Yaskawa INFORM job: SKRZYNIA_5540_-90_STOPNI_20BR.JBI

/JOB
//NAME SKRZYNIA_5540_-90_STOPNI_20BR
///FOLDERNAME 02-SKRZYNIE_JOBS
//POS
///NPOS 569,569,0,38,0,0
///TOOL 0
///POSTYPE PULSE
///PULSE
C00000=0,-52280,40443,0,6876,0
C00001=-82314,-24956,17040,-59626,-27382,-6248
C00002=-93910,-8625,17040,-59626,-43355,-6248
C00003=-98846,-1061,-42166,-80308,-57081,16120
C00004=-100452,6057,-48127,-85711,-56704,21322
C00005=-95817,31791,-34187,-84788,-63710,26674
C00006=-95573,33077,-33257,-84645,-64023,26851
C00007=-94315,33778,-32137,-85160,-63467,26714
C00008=-95573,33077,-33257,-84645,-64023,26851
C00009=-94948,31301,-36075,-85235,-63717,27152
C00010=-95573,33077,-33257,-84645,-64023,26851
C00011=-95263,33142,-33256,-84677,-63995,26850
C00012=-95263,33142,-33256,-84677,-63995,26850
C00013=-94230,33719,-32331,-85099,-63538,26735
C00014=-95263,33142,-33256,-84677,-63995,26850
C00015=-94794,31816,-35365,-85120,-63763,27076
C00016=-95263,33142,-33256,-84677,-63995,26850
C00017=-95260,33144,-33256,-84678,-63995,26850
C00018=-95260,33144,-33256,-84678,-63995,26850
C00019=-94260,33701,-32361,-85086,-63552,26738
C00020=-95260,33144,-33256,-84678,-63995,26850
C00021=-94835,31943,-35167,-85080,-63786,27056
C00022=-95260,33144,-33256,-84678,-63995,26850
C00023=-95258,25631,32269,-66559,-75499,2416
C00024=-95258,25631,32269,-66559,-75499,2416
C00025=-94256,26435,33444,-66420,-74940,2208
C00026=-95258,25631,32269,-66559,-75499,2416
C00027=-94857,24030,29962,-66606,-75105,2539
C00028=-95258,25631,32269,-66559,-75499,2416
C00029=-98811,21047,-15512,-99242,-81394,20987
C00030=-98811,21047,-15512,-99242,-81394,20987
C00031=-97856,21592,-14760,-99539,-80803,20995
C00032=-98811,21047,-15512,-99242,-81394,20987
C00033=-98487,19855,-17143,-99373,-81250,21110
C00034=-98811,21047,-15512,-99242,-81394,20987
C00035=-99077,36985,67047,-90824,-74996,11
C00036=-99077,36985,67047,-90824,-74996,11
C00037=-98126,38026,68808,-90519,-74354,-175
C00038=-99077,36985,67047,-90824,-74996,11
C00039=-98675,34279,62554,-90994,-74807,523
C00040=-99077,36985,67047,-90824,-74996,11
C00041=-98046,30065,45001,-99674,-75008,5996
C00042=-96663,27244,32711,-106417,-76052,10001
C00043=-96035,27733,33435,-106407,-75606,10011
C00044=-96663,27244,32711,-106417,-76052,10001
C00045=-96274,25568,30264,-106516,-75947,10234
C00046=-96663,27244,32711,-106417,-76052,10001
C00047=-93416,-2088,4699,-99676,-50441,9343
C00048=-88080,-20128,-3199,-80943,-31244,2335
C00049=-48287,-55439,-44481,-48508,-5390,-10469
C00050=-48287,-44591,-17414,-16172,-14532,-25809
C00051=-73855,-32171,-5678,-43952,-33220,-11069
C00052=-84843,-2315,38096,-46044,-43440,-11681
C00053=-99590,25338,21334,-81459,-78469,-3358
C00054=-99590,25338,21334,-81459,-78469,-3358
C00055=-98681,25943,22203,-81468,-77867,-3455
C00056=-99590,25338,21334,-81459,-78469,-3358
C00057=-99296,24016,19444,-81525,-78239,-3225
C00058=-99590,25338,21334,-81459,-78469,-3358
C00059=-99820,26032,21623,-82067,-78848,-4447
C00060=-99820,26032,21623,-82067,-78848,-4447
C00061=-98898,26645,22513,-82083,-78237,-4546
C00062=-99820,26032,21623,-82067,-78848,-4447
C00063=-99438,24292,19129,-82156,-78552,-4268
C00064=-99820,26032,21623,-82067,-78848,-4447
C00065=-95331,1432,-9864,-84798,-60031,-3557
C00066=-91210,-11403,-27677,-113165,-52408,5733
C00067=-98271,-15326,-41207,-114268,-59488,7673
C00068=-83743,-25164,-57719,-138536,-50905,17366
C00069=-83743,-25361,-52011,-136459,-47698,15842
C00070=-93071,-30029,-62286,-132724,-54351,14554
C00071=-61872,-66272,-83954,-148251,-32298,21081
C00072=-61872,-49557,-32264,-110357,-15428,1928
C00073=-65143,-26385,24751,-20080,-56896,-30933
C00074=-90244,4395,51028,-38516,-59607,-23032
C00075=-79356,-9150,9683,-42499,-40407,-18801
C00076=-98951,25836,42573,-74290,-75705,-4216
C00077=-99097,30513,38864,-76423,-80199,-875
C00078=-97872,31473,40332,-76298,-79437,-1085
C00079=-99097,30513,38864,-76423,-80199,-875
C00080=-98774,28880,36400,-76469,-79893,-679
C00081=-99097,30513,38864,-76423,-80199,-875
C00082=-99862,24525,29609,-86160,-76987,1407
C00083=-99452,22245,7122,-97683,-80070,9369
C00084=-99292,23987,9562,-97373,-81102,9104
C00085=-98184,24694,10564,-97522,-80343,9095
C00086=-99292,23987,9562,-97373,-81102,9104
C00087=-99030,22873,7999,-97442,-80972,9229
C00088=-99292,23987,9562,-97373,-81102,9104
C00089=-95017,-9844,-333,-79976,-47193,-2364
C00090=-62804,-32782,1918,-36164,-30925,-23493
C00091=-48283,-21883,28214,-25170,-26491,48363
C00092=-45951,-10962,51022,-17493,-32991,44756
C00093=-50347,-18571,12268,-49104,-16423,60029
C00094=-52008,-16476,13921,-52720,-16985,61589
C00095=-50839,-15356,14836,-51561,-16264,61168
C00096=-51137,-15647,14596,-51864,-16447,61279
C00097=-52695,-14846,15261,-54465,-17168,62360
C00098=-51384,-16746,13703,-51673,-16698,61154
C00099=-50347,-18571,12268,-49104,-16423,60029
C00100=-52476,-17044,12146,-55476,-16783,62883
C00101=-51467,-16091,12918,-54586,-16145,62570
C00102=-51762,-16375,12685,-54854,-16332,62665
C00103=-53129,-15664,13268,-57063,-16995,63582
C00104=-52557,-17119,12084,-55547,-16837,62908
C00105=-50509,-19000,10610,-51503,-15997,61182
C00106=-52966,-16930,12240,-56194,-17032,63176
C00107=-51879,-15912,13067,-55265,-16346,62852
C00108=-52154,-16175,12851,-55507,-16521,62938
C00109=-53227,-15612,13314,-57215,-17042,63646
C00110=-52966,-16930,12240,-56194,-17032,63176
C00111=-50703,-18403,11066,-52155,-16024,61477
C00112=-52780,-17619,11680,-55562,-17015,62889
C00113=-51306,-16241,12790,-54268,-16084,62435
C00114=-51660,-16583,12512,-54593,-16308,62551
C00115=-53327,-15718,13220,-57282,-17114,63667
C00116=-52780,-17619,11680,-55562,-17015,62889
C00117=-50704,-18401,11069,-52157,-16021,61478
C00118=-53191,-17342,11901,-56260,-17204,63181
C00119=-51773,-16022,12969,-55050,-16305,62760
C00120=-52146,-16378,12679,-55379,-16540,62876
C00121=-53214,-15820,13135,-57085,-17059,63584
C00122=-53002,-17172,12037,-56105,-17083,63128
C00123=-51005,-17995,11387,-52847,-16122,61778
C00124=-52654,-17319,11922,-55560,-16911,62904
C00125=-51372,-16113,12897,-54432,-16099,62508
C00126=-51648,-16379,12679,-54684,-16273,62598
C00127=-52952,-15703,13233,-56807,-16903,63480
C00128=-53323,-17134,12070,-56539,-17248,63304
C00129=-52826,-20105,4812,-63938,-15678,66983
C00130=-52298,-19620,5183,-63681,-15322,66914
C00131=-51076,-18450,6096,-63049,-14499,66733
C00132=-51419,-18785,5831,-63233,-14731,66786
C00133=-52680,-18133,6347,-65138,-15424,67581
C00134=-52924,-19431,7025,-60935,-16175,65505
C00135=-51752,-18759,10786,-53484,-16613,62002
C00136=-52244,-17884,11471,-54682,-16766,62529
C00137=-50303,-16031,12961,-52880,-15542,61887
C00138=-50741,-16464,12607,-53310,-15818,62044
C00139=-52416,-15612,13306,-56135,-16617,63223
C00140=-51898,-18011,11369,-54129,-16600,62301
C00141=-50945,-18019,11363,-52741,-16103,61737
C00142=-51347,-17395,11856,-53690,-16237,62152
C00143=-49990,-16073,12923,-52376,-15383,61677
C00144=-50384,-16465,12603,-52769,-15629,61822
C00145=-52066,-15616,13298,-55654,-16423,63028
C00146=-51792,-17610,11685,-54205,-16494,62350
C00147=-50945,-18019,11363,-52741,-16103,61737
C00148=-50845,-17493,11778,-52895,-15987,61824
C00149=-49521,-16191,12826,-51571,-15155,61341
C00150=-49894,-16567,12520,-51958,-15389,61484
C00151=-51728,-15654,13268,-55171,-16246,62832
C00152=-51082,-17431,11827,-53280,-16102,61986
C00153=-50028,-23690,-6096,-22921,-31075,54538
C00154=-50346,-22995,-5584,-23393,-31002,54768
C00155=-48843,-21430,-4410,-21901,-30270,54078
C00156=-49178,-21788,-4683,-22239,-30433,54235
C00157=-50538,-21100,-4158,-23908,-30654,55032
C00158=-50252,-22811,-5450,-23315,-30936,54734
C00159=-49763,-24818,-32918,-23163,-28604,59699
C00160=-49144,-24298,-32242,-22455,-28505,59304
C00161=-47766,-22458,-30816,-21237,-27774,58615
C00162=-48099,-22913,-31171,-21534,-27949,58786
C00163=-49602,-21997,-30448,-23301,-28174,59772
C00164=-49259,-23869,-32392,-22880,-28141,59533
C00165=-50713,-12366,-58367,-41124,-17813,74400
C00166=-50097,-11438,-57505,-40749,-17495,74109
C00167=-49105,-9842,-55994,-40096,-16991,73614
C00168=-49355,-10250,-56383,-40269,-17116,73742
C00169=-50506,-9357,-55529,-41571,-17503,74586
C00170=-49771,-10920,-57018,-40545,-17327,73951
C00171=-50713,-12366,-58367,-41124,-17813,74400
C00172=-50097,-11438,-57505,-40749,-17495,74109
C00173=-49105,-9842,-55994,-40096,-16991,73614
C00174=-49355,-10250,-56383,-40269,-17116,73742
C00175=-50506,-9357,-55529,-41571,-17503,74586
C00176=-49771,-10920,-57018,-40545,-17327,73951
C00177=-46548,-30139,-39639,-20061,-27197,57955
C00178=-48797,-26670,-6576,-20404,-32539,53259
C00179=-45389,-28224,4312,-35967,-15579,54278
C00180=-40154,-51179,-915,-24203,-8234,36524
C00181=0,-52280,40443,0,6876,0
C00182=-2117,-50103,-33543,-4117,45077,85249
C00183=26439,-48928,-33543,-4117,-52362,85249
C00184=26439,-27355,-33543,-41485,-52362,85249
C00185=39218,-24492,-41653,-51934,-39374,86964
C00186=38244,-2284,-24157,-56964,-37300,90090
C00187=26640,586,-20198,-77712,-51919,89712
C00188=26323,460,-20341,-77681,-52125,89737
C00189=25607,3186,-17293,-77585,-52601,89760
C00190=26323,460,-20341,-77681,-52125,89737
C00191=27719,1044,-19697,-77798,-51218,89644
C00192=26640,586,-20198,-77712,-51919,89712
C00193=46457,7101,-11330,-26648,-40775,82885
C00194=47439,8350,-9833,-26106,-40556,82449
C00195=46334,10684,-6981,-26557,-41070,82837
C00196=47439,8350,-9833,-26106,-40556,82449
C00197=48354,9159,-8854,-25603,-40343,82046
C00198=47439,8350,-9833,-26106,-40556,82449
C00199=24760,-3019,-10726,-94610,-54398,89614
C00200=25145,-1220,-8811,-94681,-54143,89655
C00201=24492,1290,-6066,-94601,-54582,89624
C00202=25145,-1220,-8811,-94681,-54143,89655
C00203=26584,-669,-8211,-94866,-53174,89734
C00204=25145,-1220,-8811,-94681,-54143,89655
C00205=14532,-15164,-22494,-92943,-61192,88617
C00206=-33377,-12679,-20251,-90012,-93751,87621
C00207=-32674,-7309,22058,-70557,-98373,80594
C00208=20046,-29908,-41690,-58842,-55822,75080
C00209=46158,10269,-6164,-23128,-46470,70172
C00210=51306,10256,-19432,-23475,-33025,71236
C00211=50386,12004,-17260,-23922,-33430,71616
C00212=51306,10256,-19432,-23475,-33025,71236
C00213=51995,10928,-18601,-23012,-32906,70879
C00214=51306,10256,-19432,-23475,-33025,71236
C00215=50667,8104,-22050,-23976,-33027,71608
C00216=27434,3323,14960,-56922,-57501,78346
C00217=29014,6574,18756,-56344,-56678,77965
C00218=28326,9009,21700,-56459,-57175,78009
C00219=29014,6574,18756,-56344,-56678,77965
C00220=30292,7183,19486,-55908,-55969,77693
C00221=29014,6574,18756,-56344,-56678,77965
C00222=24457,-1296,-8898,-94600,-54606,89622
C00223=24457,-1296,-8898,-94600,-54606,89622
C00224=23939,748,-6672,-94541,-54956,89598
C00225=24457,-1296,-8898,-94600,-54606,89622
C00226=25626,-864,-8432,-94748,-53818,89684
C00227=24457,-1296,-8898,-94600,-54606,89622
C00228=22058,-20035,-26567,-93333,-56013,88551
C00229=-28907,-25632,-31027,-90338,-90583,86609
C00230=-23923,-11573,-19230,-90501,-87328,87840
C00231=-8646,-8251,-7782,-76032,-82054,83740
C00232=42001,26537,64712,-25019,-74648,68382
C00233=42692,25604,59505,-25067,-71864,68798
C00234=42100,27723,62792,-25233,-72628,68820
C00235=42692,25604,59505,-25067,-71864,68798
C00236=43179,26157,60355,-24838,-71882,68629
C00237=42692,25604,59505,-25067,-71864,68798
C00238=42064,17796,48100,-25604,-70267,69397
C00239=28113,-7386,-15136,-95790,-47335,90009
C00240=28228,-6488,-14240,-95859,-47266,90053
C00241=27767,-5044,-12775,-95858,-47588,90072
C00242=28228,-6488,-14240,-95859,-47266,90053
C00243=29468,-5989,-13737,-96077,-46438,90154
C00244=28228,-6488,-14240,-95859,-47266,90053
C00245=51937,664,-7429,-160484,-50080,89770
C00246=52345,1107,-6938,-160727,-50007,89930
C00247=51359,2767,-5080,-160136,-50147,89540
C00248=52345,1107,-6938,-160727,-50007,89930
C00249=53054,1752,-6222,-161147,-49882,90209
C00250=52345,1107,-6938,-160727,-50007,89930
C00251=51937,664,-7429,-160484,-50080,89770
C00252=29691,-10745,-18393,-95770,-46230,89933
C00253=26663,-19279,-25970,-94307,-48104,89008
C00254=29542,-7588,-14846,-100915,-46930,90773
C00255=29616,-6902,-10165,-96183,-45225,84004
C00256=29097,-5391,-8640,-96201,-45588,84023
C00257=29616,-6902,-10165,-96183,-45225,84004
C00258=31098,-6282,-9543,-96410,-44233,84135
C00259=29616,-6902,-10165,-96183,-45225,84004
C00260=7576,-30273,-44451,-97512,-61182,86443
C00261=-18624,-40022,-50597,-93591,-78329,83668
C00262=-32134,-30783,-37092,-96173,-88064,83581
C00263=23774,-1324,-8929,-94512,-55065,89585
C00264=23774,-1324,-8929,-94512,-55065,89585
C00265=23319,517,-6924,-94461,-55372,89567
C00266=23774,-1324,-8929,-94512,-55065,89585
C00267=25077,-853,-8421,-94674,-54188,89653
C00268=23774,-1324,-8929,-94512,-55065,89585
C00269=22107,-1052,28039,-94807,-51389,77849
C00270=19995,-16885,24938,-75612,-39910,62837
///LIMIT ON
C00271=8393,-42921,36369,-24238,-5473,19544
///LIMIT OFF
C00272=0,-52280,40443,0,6876,0
C00273=-82314,-24956,17040,-59626,-27382,-6248
C00274=-93910,-8625,17040,-59626,-43355,-6248
C00275=-98846,-1061,-42166,-80308,-57081,16120
C00276=-100452,6057,-48127,-85711,-56704,21322
C00277=-95564,34698,-34234,-85516,-63941,27819
C00278=-94021,36658,-30981,-84167,-64832,27454
C00279=-93851,36773,-30815,-84181,-64812,27439
C00280=-95564,34698,-34234,-85516,-63941,27819
C00281=-96930,32282,-32252,-82595,-65816,26305
C00282=-93901,32995,-31122,-83953,-64436,26132
C00283=-93891,32978,-31150,-83961,-64431,26134
C00284=-96930,32282,-32252,-82595,-65816,26305
C00285=-97719,-4194,-31542,-76086,-54596,10626
C00286=-88377,-34186,-45291,-67238,-52212,2442
C00287=-73560,-62084,7826,-28695,-34737,-3666
C00288=0,-52280,40443,0,6876,0
C00289=0,-52280,40443,0,6876,0
C00290=-2117,-50103,-33543,-4117,45077,85249
C00291=26439,-48928,-33543,-4117,-52362,85249
C00292=26439,-27355,-33543,-41485,-52362,85249
C00293=39218,-24492,-41653,-51934,-39374,86964
C00294=37381,-5106,-22608,-53943,-39515,88347
C00295=38119,-10689,-19379,-70548,-34101,88029
C00296=37906,-14512,-22901,-69984,-34376,87713
C00297=41414,6981,-5927,-33889,-45598,86373
C00298=42289,10624,-1511,-33365,-45508,85956
C00299=42351,10656,-1473,-33340,-45486,85935
C00300=41414,6981,-5927,-33889,-45598,86373
C00301=53221,-12364,-8957,-19277,-47766,73858
C00302=11365,-15171,10010,-30164,-77975,82960
C00303=16156,-38280,11293,-23671,-42998,42040
C00304=11365,-47379,10010,-30164,3063,681
C00305=0,-52280,40443,0,6876,0
C00306=0,-36700,24612,42871,-31823,33862
C00307=-44403,-30110,7154,-24155,-23805,45557
C00308=-51570,-19542,10947,-41619,-21811,53396
C00309=-51570,-17239,16856,-38066,-23574,51584
C00310=-55052,-13712,19754,-43494,-24529,53873
C00311=-55190,-12778,21730,-42693,-25060,53437
C00312=-40431,-28773,9158,-17648,-23273,42875
C00313=0,-36700,24612,42871,-31823,33862
C00314=0,-52280,40443,0,6876,0
C00315=0,-52280,40443,0,6876,0
C00316=-73560,-62084,7826,-28695,-34737,-3666
C00317=-88377,-34186,-45291,-67238,-52212,2442
C00318=-99860,-8392,-35780,-75647,-56000,10650
C00319=-100432,21324,12575,-83706,-77956,7498
C00320=-100432,21324,12575,-83706,-77956,7498
C00321=-97477,24790,17443,-83584,-77881,7143
C00322=-97548,25214,18044,-83537,-78171,7107
C00323=-100432,21324,12575,-83706,-77956,7498
C00324=-100473,21504,12824,-83696,-77986,7482
C00325=-97708,25565,18549,-83502,-78342,7077
C00326=-97720,26100,19317,-83456,-78605,7025
C00327=-100432,21324,12575,-83706,-77956,7498
C00328=-98403,3681,-8965,-86029,-63956,7946
C00329=-98851,2841,7216,-80537,-62817,1838
C00330=-99868,-33,22146,-72719,-59601,-5126
C00331=-99028,-10516,17309,-71061,-60695,-4227
C00332=-58820,-39124,10926,-53325,-41870,-3759
C00333=0,-52280,40443,0,6876,0
C00334=-37281,-50778,-9546,-79570,-75313,71156
C00335=-21038,-23698,-30323,-82948,-81132,85647
C00336=-21230,-24252,-33397,-84866,-81311,86227
C00337=26224,-11477,-22521,-89106,-49066,87170
C00338=30473,789,4724,-68168,-47848,79016
C00339=30460,-1091,-3608,-71823,-46530,81583
C00340=26224,-11477,-22521,-89106,-49066,87170
C00341=1250,-26379,-34995,-85812,-66036,85728
C00342=-29373,-17697,-13794,-84248,-87305,82376
C00343=-12562,-22815,-22029,-52123,-75138,85349
C00344=41964,2536,-13642,-34848,-42769,74522
C00345=37974,4101,-26304,-58477,-36842,84551
C00346=37992,4823,-31618,-63468,-34913,87461
C00347=41439,5489,-14791,-37032,-40569,75962
C00348=38833,-3286,10682,-41231,-51577,69207
C00349=-9276,-22918,-17698,-90837,-69000,78700
C00350=-8172,-56778,-49528,-75726,-40055,75711
C00351=-3982,-61001,-53003,-69042,-33087,73336
C00352=37287,-55159,35520,-2191,5667,2084
C00353=0,-52280,40443,0,6876,0
C00354=0,-36700,24612,42871,-31823,33862
C00355=-44403,-30110,7154,-24155,-23805,45557
C00356=-44403,-30110,7154,-24155,-23805,45557
C00357=-42101,-12213,25656,-103795,-5192,78630
C00358=-46259,-8171,27719,-110365,-8144,81138
C00359=-67532,2461,52564,-58221,-38014,54436
C00360=-67092,2390,52438,-57975,-37749,54380
C00361=-61158,-4651,8765,-137237,-40004,88174
C00362=-56934,-15752,2926,-132390,-27589,90381
C00363=-47073,-34549,9488,-27883,-30316,51458
C00364=0,-52280,40443,0,6876,0
C00365=0,-52280,40443,0,6876,0
C00366=-73560,-62084,7826,-28695,-34737,-3666
C00367=-96366,-17217,16860,-56620,-71703,-18245
C00368=-98152,-14905,2044,-65675,-67485,-3494
C00369=-100467,-7393,-15195,-81625,-60158,6002
C00370=-99336,18440,8642,-84276,-74234,7647
C00371=-99336,18440,8642,-84276,-74234,7647
C00372=-97907,25479,18429,-83510,-78268,7080
C00373=-97774,25771,18838,-83486,-78362,7054
C00374=-99336,18440,8642,-84276,-74234,7647
C00375=-99336,20364,19482,-82786,-74642,4774
C00376=-98337,25059,18813,-87846,-78771,10707
C00377=-98337,23926,10585,-88652,-78855,12971
C00378=-99528,19847,13673,-83665,-74506,6500
C00379=-89817,-17341,-38408,-97132,-45323,12250
C00380=-100347,-21961,-42251,-93939,-52125,11121
C00381=-60204,-59872,-73451,-117647,-17639,18840
C00382=-37721,-67612,11381,-1325,-438,-7850
C00383=0,-52280,40443,0,6876,0
C00384=37287,-55159,35520,-2191,5667,2084
C00385=40042,-68802,-18337,-47708,-19461,45384
C00386=16481,-63411,-38742,-86271,-37962,67106
C00387=28646,-23138,-32952,-89786,-42552,85395
C00388=38882,-16596,-17625,-44304,-41043,72768
C00389=40930,-6862,-13364,-47045,-37020,74415
C00390=41744,-3361,-9781,-46774,-36492,74231
C00391=41678,-4243,-16493,-50979,-33997,76666
C00392=40930,-6862,-13364,-47045,-37020,74415
C00393=38882,-16596,-17625,-44304,-41043,72768
C00394=28646,-23138,-32952,-89786,-42552,85395
C00395=29905,-15291,-26411,-91102,-43435,86304
C00396=31540,-7654,-19248,-92177,-42391,86919
C00397=31445,-8095,-22888,-97196,-43117,89457
C00398=29637,-16450,-35189,-96198,-44206,89682
C00399=-7164,-46429,-55577,-86274,-68578,84143
C00400=40042,-68802,-18337,-47708,-19461,45384
C00401=37287,-55159,35520,-2191,5667,2084
C00402=0,-52280,40443,0,6876,0
C00403=-37164,-60659,6466,-13301,-5027,19773
C00404=-45362,-39990,2831,-27538,-17767,40935
C00405=-57189,-26834,-7130,-38780,-31731,51561
C00406=-55974,-20661,-3180,-39617,-29741,52134
C00407=-55991,-28453,-45977,-64163,-20900,63765
C00408=-57189,-26834,-7130,-38780,-31731,51561
C00409=-41180,-61187,4729,-17280,-8498,23442
C00410=0,-52280,40443,0,6876,0
C00411=0,-52280,40443,0,6876,0
C00412=-43180,-50572,-20637,-6552,-29302,-38834
C00413=-79425,-37128,-15462,-51820,-35721,-18807
C00414=-93702,-21743,-5664,-65079,-41536,-12324
C00415=-94876,-11469,-23586,-124528,-59237,5423
C00416=-92861,23404,17376,-116518,-76732,-1573
C00417=-96665,29896,42633,-98437,-75635,-11031
C00418=-96665,37701,65506,-96077,-73868,-15674
C00419=-98256,26642,30161,-104402,-77650,-7294
C00420=-94876,-11469,-23586,-124528,-59237,5423
C00421=-94108,-26192,-19530,-80749,-38523,-6311
C00422=-79425,-37128,-15462,-51820,-35721,-18807
C00423=-44920,-50063,-20090,-8739,-29356,-37564
C00424=-37721,-67612,11381,-1325,-438,-7850
C00425=0,-52280,40443,0,6876,0
C00426=40043,-68802,-18337,-47706,-19461,45383
C00427=27078,-46675,7729,-35821,-60236,53359
C00428=37661,6027,34279,-36092,-58837,68690
C00429=38848,9668,32452,-36978,-55195,69693
C00430=45203,15557,41040,-24527,-60177,66840
C00431=37661,2340,23735,-37788,-55306,70200
C00432=22173,-30639,7984,-58136,-45615,60133
C00433=37287,-55159,35520,-2191,5667,2084
C00434=0,-52280,40443,0,6876,0
C00435=-23708,-46776,23536,-16027,-4787,19738
C00436=-50917,-40459,4132,-34421,-18173,42391
C00437=-54964,-26842,8528,-44141,-23181,52038
C00438=-51719,-20944,8196,-48593,-18539,54728
C00439=-53338,-16066,12564,-52314,-18938,56375
C00440=-53668,-14237,17353,-48629,-20286,54493
C00441=-18010,-41727,-5437,24633,-20435,23511
C00442=-18010,-41727,-5437,24633,-20435,23511
C00443=-43180,-50572,-20637,-6552,-29302,-38834
C00444=-37721,-67612,11381,-1325,-438,-7850
C00445=0,-52280,40443,0,6876,0
C00446=-7830,-25136,17099,-55306,-64068,52084
C00447=34592,-23156,18291,-29932,-45204,43222
C00448=27626,-5609,7480,-74303,-46810,69713
C00449=30162,-7263,-3756,-79871,-43922,73611
C00450=30945,-3557,12,-79972,-43367,73694
C00451=30934,-3652,-86,-79966,-43372,73693
C00452=29106,-7674,-4162,-79972,-44640,73655
C00453=-2837,-32019,-23857,-80741,-66785,72567
C00454=9534,-43450,13514,-26959,-29486,38723
C00455=22834,-59963,22946,-6692,-2150,9612
C00456=0,-52280,40443,0,6876,0
C00457=-23708,-46776,23536,-16027,-4787,19738
C00458=-50917,-40459,4132,-34421,-18173,42391
C00459=-51059,-36587,4608,-36647,-19418,45358
C00460=-50113,-22729,10834,-36393,-23396,50963
C00461=-57831,-20321,-874,-74195,-20905,72937
C00462=-57885,-15500,12470,-61600,-22854,66553
C00463=-50113,-22729,10834,-36393,-23396,50963
C00464=-45969,-44671,-42317,80322,10570,10889
C00465=-31285,-69981,-10849,-7246,-6842,20992
C00466=0,-52280,40443,0,6876,0
C00467=-37721,-67612,11381,-1325,-438,-7850
C00468=-43180,-50572,-20637,-6552,-29302,-38834
C00469=-92181,-6909,34626,-50562,-49190,-21840
C00470=-101117,-5694,-18308,-85789,-60825,2377
C00471=-97622,-3602,-16155,-86160,-58465,2400
C00472=-99754,24347,18348,-83049,-78046,1543
C00473=-98401,23935,17754,-83131,-77323,1564
C00474=-98274,24050,17917,-83129,-77329,1551
C00475=-99954,24418,19993,-82828,-78557,1051
C00476=-99712,24798,18984,-83012,-78332,1506
C00477=-99852,25442,19906,-82977,-78439,1439
C00478=-98294,26390,21274,-82926,-78604,1336
C00479=-98320,27540,23370,-82787,-79202,1083
C00480=-99852,25442,19906,-82977,-78439,1439
C00481=-99768,8894,-2445,-89351,-68751,3793
C00482=-96099,-3787,-16815,-92200,-58195,4535
C00483=-97559,-25159,-36085,-93407,-46496,3918
C00484=-68601,-52593,-52127,-95725,-25602,3235
C00485=-80632,-38079,-20908,-64053,-45216,-12949
C00486=-43180,-50572,-20637,-6552,-29302,-38834
///LIMIT ON
C00487=-37721,-67612,11381,-1325,-438,-7850
///LIMIT OFF
C00488=54026,-30203,28811,7745,-28969,5087
C00489=55906,-29650,27841,6704,-28568,42061
C00490=3910,-49110,-20873,-64325,-51391,71742
C00491=9596,-41005,-15480,-61992,-50741,70573
C00492=34629,-5327,8260,-51720,-47880,65426
C00493=35679,2837,17551,-51053,-47466,65038
C00494=35689,-56,7549,-54586,-44718,67469
C00495=34629,-5327,8260,-51720,-47880,65426
C00496=9596,-41005,-15480,-61992,-50741,70573
C00497=29660,-4584,-26917,-122917,-59269,85605
C00498=30458,-1431,-23593,-123278,-58903,85810
C00499=32051,-581,-21149,-126899,-58917,85995
C00500=28378,-5181,-30467,-124970,-61925,86269
C00501=9596,-41005,-15480,-61992,-50741,70573
C00502=4124,-42500,-16101,-63937,-54198,71061
C00503=22834,-59963,22946,-6692,-2150,9612
C00504=0,-52280,40443,0,6876,0
C00505=-44101,-76445,-48847,-15697,-17168,40457
C00506=-48984,-30078,-36716,-21434,-29637,58750
C00507=-50484,-13386,-55713,-36158,-19724,71897
C00508=-50319,-9696,-53018,-37576,-18929,72579
C00509=-57729,15185,-57220,-77412,-21272,89270
C00510=-57753,15208,-57190,-77395,-21282,89267
C00511=-50484,-13386,-55713,-36158,-19724,71897
C00512=-49763,-25421,-36239,-24565,-26935,60445
C00513=-50529,-22709,-3778,-22940,-31995,54502
C00514=-45389,-28224,4312,-35967,-15579,54278
C00515=-40154,-51179,-915,-24203,-8234,36524
C00516=0,-52280,40443,0,6876,0
C00517=0,-52280,40443,0,6876,0
///LIMIT ON
C00518=-37721,-67612,11381,-1325,-438,-7850
///LIMIT OFF
C00519=-43180,-50572,-20637,-6552,-29302,-38834
C00520=-43180,-50572,-20637,-6552,-29302,-38834
C00521=-91233,-13472,9135,-57436,-42793,-15671
C00522=-94453,18451,26397,-64403,-69695,-4898
C00523=-94848,25710,19994,-67599,-74328,1083
C00524=-94734,25454,19627,-67614,-74234,1097
C00525=-94605,24228,10738,-68938,-72404,3439
C00526=-96555,21614,11724,-68276,-72695,2131
C00527=-99000,22482,23037,-75261,-76004,639
C00528=-97210,28604,31066,-74659,-78513,378
C00529=-97154,26647,21384,-75593,-77346,2770
C00530=-100531,16612,13557,-75306,-72509,1088
C00531=-98914,15791,22093,-91892,-69242,2220
C00532=-98524,31242,37673,-92432,-80087,2200
C00533=-98508,35203,51300,-91477,-79539,-794
C00534=-99299,29399,42249,-91532,-77608,155
C00535=-99299,39874,71997,-89061,-76925,-5800
C00536=-98153,38420,66100,-91432,-76531,-4068
C00537=-98147,36464,60868,-91873,-76694,-3060
C00538=-99718,12303,6039,-96207,-71156,6635
C00539=-93032,-8711,-3060,-81304,-48072,-4095
C00540=-98228,-14972,-11291,-81392,-49231,-4002
C00541=-91129,-17870,8831,-66292,-48444,-14183
C00542=-68865,-35989,-5252,-49829,-38105,-21179
C00543=-15566,-52364,-9989,12732,-35649,-46896
C00544=0,-52278,40443,-31822,-65283,46097
C00545=7820,3000,44222,-77356,-66876,70486
C00546=23103,22769,71034,-65639,-61603,67373
C00547=25078,30713,84198,-63240,-61811,65668
C00548=25008,30264,83410,-63369,-61766,65773
C00549=23103,22769,71034,-65639,-61603,67373
C00550=23103,22769,71034,-65639,-61603,67373
C00551=25078,30713,84198,-63240,-61811,65668
C00552=25008,30264,83410,-63369,-61766,65773
C00553=23103,22769,71034,-65639,-61603,67373
C00554=-3014,-20441,-7349,-104591,-68614,79454
C00555=-3014,-20441,-7349,-104591,-68614,79454
C00556=-13238,-21720,-1359,-93359,-59492,72612
C00557=10261,-46634,14475,-36899,-22136,31570
///LIMIT ON
C00558=22834,-59963,22946,-6692,-2150,9612
///LIMIT OFF
C00559=0,-52280,40443,0,6876,0
///LIMIT ON
C00560=-23708,-46776,23536,-16027,-4787,19738
///LIMIT OFF
C00561=-50917,-40459,4132,-34421,-18173,42391
C00562=-49876,-21948,7530,-68838,-10324,59148
C00563=-46721,-18942,9765,-68167,-8197,59205
C00564=-47628,-14741,12915,-75746,-8483,62696
C00565=-48046,-13368,16308,-68442,-9096,59180
C00566=-42573,-24036,4541,-56448,-5917,54155
C00567=-31287,-69981,-10850,-7253,-6843,20996
C00568=0,-52280,40443,0,6876,0
BC00000=471249
BC00001=460491
BC00002=460491
BC00003=460491
BC00004=460491
BC00005=482540
BC00006=483588
BC00007=483588
BC00008=483588
BC00009=483588
BC00010=483588
BC00011=529782
BC00012=529782
BC00013=529782
BC00014=529782
BC00015=529782
BC00016=529782
BC00017=575949
BC00018=575949
BC00019=575949
BC00020=575949
BC00021=575949
BC00022=575949
BC00023=551765
BC00024=551765
BC00025=551765
BC00026=551765
BC00027=551765
BC00028=551765
BC00029=597819
BC00030=597819
BC00031=597819
BC00032=597819
BC00033=597819
BC00034=597819
BC00035=596567
BC00036=596567
BC00037=596567
BC00038=596567
BC00039=596567
BC00040=596567
BC00041=623804
BC00042=642102
BC00043=642102
BC00044=642102
BC00045=642102
BC00046=642102
BC00047=619616
BC00048=619616
BC00049=642599
BC00050=714482
BC00051=745522
BC00052=745522
BC00053=836176
BC00054=836176
BC00055=836176
BC00056=836176
BC00057=836176
BC00058=836176
BC00059=881624
BC00060=881624
BC00061=881624
BC00062=881624
BC00063=881624
BC00064=881624
BC00065=881624
BC00066=887605
BC00067=887605
BC00068=887605
BC00069=887605
BC00070=887605
BC00071=887605
BC00072=887605
BC00073=983293
BC00074=981254
BC00075=985702
BC00076=990046
BC00077=996594
BC00078=996594
BC00079=996594
BC00080=996594
BC00081=996594
BC00082=994630
BC00083=1060317
BC00084=1060317
BC00085=1060317
BC00086=1060317
BC00087=1060317
BC00088=1060317
BC00089=993852
BC00090=983691
BC00091=935062
BC00092=958518
BC00093=1027445
BC00094=1027445
BC00095=1027445
BC00096=1027445
BC00097=1027445
BC00098=1027445
BC00099=964364
BC00100=968743
BC00101=968743
BC00102=968743
BC00103=968743
BC00104=968743
BC00105=903417
BC00106=903417
BC00107=903417
BC00108=903417
BC00109=903417
BC00110=903417
BC00111=846075
BC00112=846075
BC00113=846075
BC00114=846075
BC00115=846075
BC00116=846075
BC00117=780190
BC00118=780190
BC00119=780190
BC00120=780190
BC00121=780190
BC00122=780190
BC00123=722535
BC00124=722535
BC00125=722535
BC00126=722535
BC00127=722535
BC00128=722535
BC00129=657432
BC00130=657432
BC00131=657432
BC00132=657432
BC00133=657432
BC00134=657432
BC00135=600107
BC00136=600107
BC00137=600107
BC00138=600107
BC00139=600107
BC00140=600107
BC00141=534593
BC00142=534593
BC00143=534593
BC00144=534593
BC00145=534593
BC00146=534593
BC00147=477174
BC00148=477174
BC00149=477174
BC00150=477174
BC00151=477174
BC00152=477174
BC00153=474905
BC00154=474905
BC00155=474905
BC00156=474905
BC00157=474905
BC00158=474905
BC00159=474905
BC00160=474905
BC00161=474905
BC00162=474905
BC00163=474905
BC00164=474905
BC00165=474905
BC00166=474905
BC00167=474905
BC00168=474905
BC00169=474905
BC00170=474905
BC00171=428822
BC00172=428822
BC00173=428822
BC00174=428822
BC00175=428822
BC00176=428822
BC00177=474905
BC00178=474905
BC00179=474901
BC00180=548577
BC00181=548577
BC00182=423885
BC00183=423885
BC00184=423885
BC00185=423885
BC00186=423885
BC00187=423882
BC00188=423882
BC00189=423882
BC00190=423882
BC00191=423882
BC00192=423882
BC00193=517447
BC00194=516208
BC00195=516208
BC00196=516208
BC00197=516208
BC00198=516208
BC00199=462401
BC00200=462401
BC00201=462401
BC00202=462401
BC00203=462401
BC00204=462401
BC00205=462401
BC00206=462401
BC00207=581968
BC00208=647467
BC00209=647467
BC00210=647467
BC00211=647467
BC00212=647467
BC00213=647467
BC00214=647467
BC00215=647467
BC00216=600589
BC00217=600589
BC00218=600589
BC00219=600589
BC00220=600589
BC00221=600589
BC00222=646713
BC00223=646713
BC00224=646713
BC00225=646713
BC00226=646713
BC00227=646713
BC00228=646713
BC00229=646713
BC00230=703926
BC00231=764819
BC00232=734650
BC00233=734650
BC00234=734650
BC00235=734650
BC00236=734650
BC00237=734650
BC00238=734650
BC00239=762000
BC00240=762000
BC00241=762000
BC00242=762000
BC00243=762000
BC00244=762000
BC00245=768744
BC00246=768744
BC00247=768744
BC00248=768744
BC00249=768744
BC00250=768744
BC00251=768744
BC00252=762000
BC00253=762000
BC00254=869424
BC00255=869424
BC00256=869424
BC00257=869424
BC00258=869424
BC00259=869424
BC00260=869424
BC00261=869424
BC00262=983898
BC00263=992364
BC00264=992364
BC00265=992364
BC00266=992364
BC00267=992364
BC00268=992364
BC00269=927243
BC00270=910363
BC00271=869677
BC00272=473857
BC00273=460491
BC00274=460491
BC00275=460491
BC00276=460491
BC00277=491299
BC00278=491278
BC00279=483675
BC00280=491299
BC00281=530690
BC00282=530690
BC00283=523662
BC00284=530690
BC00285=557568
BC00286=557568
BC00287=557568
BC00288=542207
BC00289=492150
BC00290=423885
BC00291=423885
BC00292=423885
BC00293=423885
BC00294=418215
BC00295=406365
BC00296=406365
BC00297=507950
BC00298=507950
BC00299=500226
BC00300=507950
BC00301=493160
BC00302=493160
BC00303=493160
BC00304=493160
BC00305=493160
BC00306=598171
BC00307=670543
BC00308=729889
BC00309=728141
BC00310=728141
BC00311=789114
BC00312=789114
BC00313=598171
BC00314=556285
BC00315=557568
BC00316=557568
BC00317=557568
BC00318=606305
BC00319=559125
BC00320=474638
BC00321=474638
BC00322=467026
BC00323=474638
BC00324=536109
BC00325=536109
BC00326=543656
BC00327=536109
BC00328=539958
BC00329=628234
BC00330=599778
BC00331=599778
BC00332=599778
BC00333=599778
BC00334=542360
BC00335=599440
BC00336=482963
BC00337=482963
BC00338=482963
BC00339=482963
BC00340=482963
BC00341=482963
BC00342=482963
BC00343=633179
BC00344=633182
BC00345=633182
BC00346=633182
BC00347=633182
BC00348=590162
BC00349=577838
BC00350=565789
BC00351=612529
BC00352=620193
BC00353=620193
BC00354=828164
BC00355=903144
BC00356=942427
BC00357=909055
BC00358=930245
BC00359=950170
BC00360=1007113
BC00361=1029951
BC00362=961342
BC00363=868420
BC00364=557568
BC00365=557568
BC00366=528880
BC00367=572227
BC00368=592163
BC00369=606305
BC00370=587350
BC00371=582221
BC00372=582227
BC00373=588358
BC00374=582221
BC00375=641167
BC00376=648252
BC00377=646780
BC00378=643131
BC00379=650479
BC00380=650479
BC00381=648520
BC00382=733103
BC00383=733103
BC00384=620193
BC00385=620193
BC00386=625652
BC00387=635598
BC00388=635598
BC00389=635598
BC00390=635598
BC00391=635598
BC00392=635598
BC00393=635598
BC00394=635598
BC00395=658627
BC00396=658630
BC00397=665879
BC00398=658627
BC00399=658627
BC00400=620193
BC00401=620193
BC00402=620193
BC00403=561542
BC00404=498768
BC00405=467432
BC00406=467432
BC00407=467432
BC00408=467432
BC00409=539526
BC00410=539526
BC00411=748464
BC00412=748464
BC00413=630778
BC00414=630772
BC00415=630772
BC00416=630772
BC00417=638952
BC00418=638952
BC00419=636403
BC00420=630772
BC00421=630772
BC00422=652282
BC00423=713933
BC00424=733103
BC00425=733103
BC00426=667407
BC00427=721208
BC00428=721208
BC00429=721208
BC00430=727232
BC00431=730010
BC00432=686453
BC00433=620193
BC00434=620193
BC00435=576077
BC00436=557154
BC00437=596115
BC00438=604917
BC00439=604794
BC00440=662711
BC00441=664655
BC00442=784947
BC00443=795297
BC00444=733103
BC00445=733103
BC00446=727492
BC00447=727492
BC00448=759331
BC00449=759331
BC00450=759331
BC00451=766564
BC00452=759331
BC00453=759331
BC00454=672725
BC00455=672725
BC00456=672725
BC00457=766882
BC00458=806462
BC00459=818228
BC00460=851878
BC00461=860102
BC00462=909902
BC00463=851878
BC00464=813387
BC00465=767805
BC00466=733103
BC00467=733103
BC00468=748464
BC00469=748464
BC00470=831036
BC00471=832865
BC00472=832865
BC00473=832865
BC00474=839696
BC00475=839696
BC00476=877964
BC00477=878266
BC00478=878754
BC00479=885787
BC00480=878266
BC00481=840209
BC00482=834137
BC00483=827396
BC00484=765830
BC00485=798734
BC00486=810658
BC00487=748464
BC00488=762701
BC00489=765633
BC00490=830967
BC00491=835024
BC00492=852883
BC00493=852883
BC00494=852883
BC00495=852883
BC00496=835024
BC00497=861491
BC00498=861491
BC00499=861491
BC00500=861491
BC00501=835024
BC00502=835024
BC00503=672725
BC00504=672725
BC00505=543617
BC00506=474905
BC00507=474905
BC00508=474905
BC00509=459544
BC00510=450616
BC00511=474905
BC00512=474905
BC00513=474905
BC00514=474901
BC00515=548577
BC00516=548577
BC00517=748464
BC00518=748464
BC00519=869948
BC00520=986791
BC00521=981739
BC00522=1008171
BC00523=1008171
BC00524=1008171
BC00525=1008171
BC00526=1008171
BC00527=1008171
BC00528=1008171
BC00529=1008171
BC00530=1006011
BC00531=1030226
BC00532=1030226
BC00533=1030226
BC00534=1030226
BC00535=1030226
BC00536=1030226
BC00537=1042625
BC00538=1042625
BC00539=995149
BC00540=992199
BC00541=972060
BC00542=967683
BC00543=967683
BC00544=921533
BC00545=921533
BC00546=946591
BC00547=946591
BC00548=953713
BC00549=946591
BC00550=997282
BC00551=997282
BC00552=1004404
BC00553=997282
BC00554=1013986
BC00555=963295
BC00556=908449
BC00557=770245
BC00558=688086
BC00559=688086
BC00560=577701
BC00561=467723
BC00562=467723
BC00563=467723
BC00564=467723
BC00565=526528
BC00566=527247
BC00567=757643
BC00568=757643
///POSTYPE BASE
///RECTAN
///RCONF 0,0,0,0,0,0,0,0,0,0,0,0,0,0,0,0,0,0,0,0,0,0,0,0
P00006=-2.449,0.031,8.825,0.0000,0.0000,0.0000
///RCONF 1,0,0,0,0,0,0,0,0,0,0,0,0,0,0,0,0,0,0,0,0,0,0,0
P00300=-0.036,-1.505,2.318,0.0000,0.0000,0.0000
///RCONF 0,0,0,0,0,0,0,0,0,0,0,0,0,0,0,0,0,0,0,0,0,0,0,0
P00301=0.005,-4.708,-4.628,0.0000,0.0000,0.0000
P00302=0.052,-2.937,-4.426,0.0000,0.0000,0.0000
P00303=-0.004,-1.437,-4.584,0.0000,0.0000,0.0000
P00304=0.028,-1.666,-4.234,0.0000,0.0000,0.0000
P00305=-0.003,-1.920,-3.501,0.0000,0.0000,0.0000
P00306=0.015,-2.252,-3.054,0.0000,0.0000,0.0000
P00308=-0.003,-2.092,-4.888,0.0000,0.0000,0.0000
P00309=-0.040,-2.205,-4.992,0.0000,0.0000,0.0000
P00311=-0.007,-2.079,-5.307,0.0000,0.0000,0.0000
P00312=-0.032,2.202,-7.632,0.0000,0.0000,0.0000
///RCONF 1,0,0,0,0,0,0,0,0,0,0,0,0,0,0,0,0,0,0,0,0,0,0,0
P00349=0.060,0.167,-1.133,0.0000,0.0000,0.0000
///RCONF 0,0,0,0,0,0,0,0,0,0,0,0,0,0,0,0,0,0,0,0,0,0,0,0
P00350=11.519,-0.008,1.149,0.0000,0.0000,0.0000
P00351=13.563,-0.027,-0.653,0.0000,0.0000,0.0000
P00352=13.252,-0.027,-0.827,0.0000,0.0000,0.0000
P00353=10.971,-0.082,0.776,0.0000,0.0000,0.0000
P00354=-0.024,2.508,-1.824,0.0000,0.0000,0.0000
P00355=-0.001,2.528,-1.131,0.0000,0.0000,0.0000
P00356=-0.034,2.921,-0.262,0.0000,0.0000,0.0000
P00357=0.003,3.386,-0.091,0.0000,0.0000,0.0000
P00358=0.014,3.037,-0.020,0.0000,0.0000,0.0000
P00359=-0.005,2.731,0.912,0.0000,0.0000,0.0000
P00360=-0.011,3.412,0.438,0.0000,0.0000,0.0000
P00361=0.018,3.050,1.253,0.0000,0.0000,0.0000
P00362=0.014,2.784,0.148,0.0000,0.0000,0.0000
P00400=5.920,-3.503,-0.024,0.0000,0.0000,0.0000
P00401=3.430,-0.021,1.131,0.0000,0.0000,0.0000
P00402=-0.253,1.107,3.062,0.0000,0.0000,0.0000
P00403=-3.666,-0.015,5.328,0.0000,0.0000,0.0000
///RCONF 1,0,0,0,0,0,0,0,0,0,0,0,0,0,0,0,0,0,0,0,0,0,0,0
P00404=0.029,4.189,-1.030,0.0000,0.0000,0.0000
///RCONF 0,0,0,0,0,0,0,0,0,0,0,0,0,0,0,0,0,0,0,0,0,0,0,0
P00405=2.420,0.007,1.427,0.0000,0.0000,0.0000
P00406=3.513,-0.022,0.429,0.0000,0.0000,0.0000
///RCONF 1,0,0,0,1,0,0,0,0,0,0,0,0,0,0,0,0,0,0,0,0,0,0,0
P00407=-0.029,2.348,-1.469,0.0000,0.0000,0.0000
P00408=0.010,1.346,-1.479,0.0000,0.0000,0.0000
///RCONF 1,0,0,0,0,0,0,0,0,0,0,0,0,0,0,0,0,0,0,0,0,0,0,0
P00409=-0.026,2.090,-1.483,0.0000,0.0000,0.0000
P00410=0.001,4.491,-0.583,0.0000,0.0000,0.0000
///RCONF 1,0,0,0,1,0,0,0,0,0,0,0,0,0,0,0,0,0,0,0,0,0,0,0
P00411=-0.015,3.627,0.872,0.0000,0.0000,0.0000
//INST
///DATE 2025/02/25 14:00
///ATTR SC,RW
///GROUP1 RB1,BS1
NOP
CALL JOB:MOVE_INTO_TUNNEL
MOVJ C00000 BC00000 VJ=30.00
MOVJ C00001 BC00001 VJ=30.00
MOVJ C00002 BC00002 VJ=30.00
MOVL C00003 BC00003 V=500.0
MOVJ C00004 BC00004 VJ=20.00
'------------------------
'W65.3
'------------------------
MOVL C00005 BC00005 V=333.3
MOVL C00006 BC00006 V=166.7 PL=0
REFP 3 C00007 BC00007
CALL JOB:SEARCH-R1
SET P0300 P0006
SFTON P0300
MOVL C00008 BC00008 V=66.7 PL=0
REFP 3 C00009 BC00009
CALL JOB:SEARCH-R1
SET P0300 P0006
SFTON P0300
MOVL C00010 BC00010 V=66.7 PL=0
SFTOF
'------------------------
'W65.5
'------------------------
MOVL C00011 BC00011 V=500.0
MOVL C00012 BC00012 V=166.7 PL=0
REFP 3 C00013 BC00013
CALL JOB:SEARCH-R1
SET P0301 P0006
SFTON P0301
MOVL C00014 BC00014 V=166.7 PL=0
REFP 3 C00015 BC00015
CALL JOB:SEARCH-R1
SET P0301 P0006
SFTON P0301
MOVL C00016 BC00016 V=166.7 PL=0
SFTOF
'------------------------
'W65.7
'------------------------
MOVL C00017 BC00017 V=500.0
MOVL C00018 BC00018 V=166.7 PL=0
REFP 3 C00019 BC00019
CALL JOB:SEARCH-R1
SET P0302 P0006
SFTON P0302
MOVL C00020 BC00020 V=166.7 PL=0
REFP 3 C00021 BC00021
CALL JOB:SEARCH-R1
SET P0302 P0006
SFTON P0302
MOVL C00022 BC00022 V=166.7 PL=0
SFTOF
'------------------------
'W65.10
'------------------------
MOVL C00023 BC00023 V=500.0
MOVL C00024 BC00024 V=166.7 PL=0
REFP 3 C00025 BC00025
CALL JOB:SEARCH-R1
SET P0303 P0006
SFTON P0303
MOVL C00026 BC00026 V=166.7 PL=0
REFP 3 C00027 BC00027
CALL JOB:SEARCH-R1
SET P0303 P0006
SFTON P0303
MOVL C00028 BC00028 V=166.7 PL=0
SFTOF
'------------------------
'W65.12
'------------------------
MOVL C00029 BC00029 V=500.0
MOVL C00030 BC00030 V=166.7 PL=0
REFP 3 C00031 BC00031
CALL JOB:SEARCH-R1
SET P0304 P0006
SFTON P0304
MOVL C00032 BC00032 V=166.7 PL=0
REFP 3 C00033 BC00033
CALL JOB:SEARCH-R1
SET P0304 P0006
SFTON P0304
MOVL C00034 BC00034 V=166.7 PL=0
SFTOF
'------------------------
'W65.15
'------------------------
MOVL C00035 BC00035 V=333.3
MOVL C00036 BC00036 V=166.7 PL=0
REFP 3 C00037 BC00037
CALL JOB:SEARCH-R1
SET P0305 P0006
SFTON P0305
MOVL C00038 BC00038 V=166.7 PL=0
REFP 3 C00039 BC00039
CALL JOB:SEARCH-R1
SET P0305 P0006
SFTON P0305
MOVL C00040 BC00040 V=166.7 PL=0
SFTOF
'------------------------
'W65.17
'------------------------
MOVL C00041 BC00041 V=333.3
MOVL C00042 BC00042 V=166.7 PL=0
REFP 3 C00043 BC00043
CALL JOB:SEARCH-R1
SET P0306 P0006
SFTON P0306
MOVL C00044 BC00044 V=166.7 PL=0
REFP 3 C00045 BC00045
CALL JOB:SEARCH-R1
SET P0306 P0006
SFTON P0306
MOVL C00046 BC00046 V=166.7 PL=0
SFTOF
MOVL C00047 BC00047 V=333.3
MOVL C00048 BC00048 V=500.0
MOVL C00049 BC00049 V=500.0
MOVJ C00050 BC00050 VJ=50.00
MOVL C00051 BC00051 V=500.0
MOVL C00052 BC00052 V=500.0
'------------------------
'W65.20
'------------------------
'------------------------
MOVL C00053 BC00053 V=333.3
MOVL C00054 BC00054 V=166.7 PL=0
REFP 3 C00055 BC00055
CALL JOB:SEARCH-R1
SET P0308 P0006
SFTON P0308
MOVL C00056 BC00056 V=166.7 PL=0
REFP 3 C00057 BC00057
CALL JOB:SEARCH-R1
SET P0308 P0006
SFTON P0308
MOVL C00058 BC00058 V=166.7 PL=0
SFTOF
'------------------------
'W65.25
'------------------------
MOVL C00059 BC00059 V=500.0
MOVL C00060 BC00060 V=166.7 PL=0
REFP 3 C00061 BC00061
CALL JOB:SEARCH-R1
SET P0309 P0006
SFTON P0309
MOVL C00062 BC00062 V=166.7 PL=0
REFP 3 C00063 BC00063
CALL JOB:SEARCH-R1
SET P0309 P0006
SFTON P0309
MOVL C00064 BC00064 V=166.7 PL=0
SFTOF
MOVL C00065 BC00065 V=166.7
MOVL C00066 BC00066 V=666.7
MOVL C00067 BC00067 V=666.7
MOVL C00068 BC00068 V=666.7
MOVL C00069 BC00069 V=666.7
MOVL C00070 BC00070 V=666.7
MOVL C00071 BC00071 V=666.7
MOVL C00072 BC00072 V=666.7
MOVL C00073 BC00073 V=666.7
MOVL C00074 BC00074 V=666.7
MOVL C00075 BC00075 V=666.7
'------------------------
'W65.28
'------------------------
'W65.30
'------------------------
MOVL C00076 BC00076 V=500.0
MOVL C00077 BC00077 V=166.7 PL=0
REFP 3 C00078 BC00078
CALL JOB:SEARCH-R1
SET P0311 P0006
SFTON P0311
MOVL C00079 BC00079 V=166.7 PL=0
REFP 3 C00080 BC00080
CALL JOB:SEARCH-R1
SET P0311 P0006
SFTON P0311
MOVL C00081 BC00081 V=166.7 PL=0
SFTOF
MOVL C00082 BC00082 V=333.3
MOVL C00083 BC00083 V=333.3
MOVL C00084 BC00084 V=166.7
REFP 3 C00085 BC00085
CALL JOB:SEARCH-R1
SET P0312 P0006
SFTON P0312
MOVL C00086 BC00086 V=166.7 PL=0
REFP 3 C00087 BC00087
CALL JOB:SEARCH-R1
SET P0312 P0006
SFTON P0312
MOVL C00088 BC00088 V=166.7 PL=0
SFTOF
MOVL C00089 BC00089 V=333.3
MOVL C00090 BC00090 V=333.3
MOVJ C00091 BC00091 VJ=30.00
MOVJ C00092 BC00092 VJ=30.00
MOVL C00093 BC00093 V=500.0
SFTOF
MOVL C00094 BC00094 V=166.7 PL=0
REFP 3 C00095 BC00095
CALL JOB:SEARCH-R1
SET P0349 P0006
SFTON P0349
MOVL C00096 BC00096 V=166.7 PL=0
REFP 3 C00097 BC00097
CALL JOB:SEARCH-R1
SET P0349 P0006
SFTON P0349
MOVL C00098 BC00098 V=166.7 PL=0
SFTOF
MOVL C00099 BC00099 V=333.3
SFTOF
'------------------------
'W251A
'------------------------
MOVL C00100 BC00100 V=166.7 PL=0
REFP 3 C00101 BC00101
CALL JOB:SEARCH-R1
SET P0350 P0006
SFTON P0350
MOVL C00102 BC00102 V=166.7 PL=0
REFP 3 C00103 BC00103
CALL JOB:SEARCH-R1
SET P0350 P0006
SFTON P0350
MOVL C00104 BC00104 V=166.7 PL=0
SFTOF
'------------------------
'W254A P
'------------------------
MOVJ C00105 BC00105 VJ=40.00
MOVL C00106 BC00106 V=166.7 PL=0
REFP 3 C00107 BC00107
CALL JOB:SEARCH-R1
SET P0351 P0006
SFTON P0351
MOVL C00108 BC00108 V=166.7 PL=0
REFP 3 C00109 BC00109
CALL JOB:SEARCH-R1
SET P0351 P0006
SFTON P0351
MOVL C00110 BC00110 V=166.7 PL=0
SFTOF
'------------------------
'W254A L
'------------------------
MOVJ C00111 BC00111 VJ=40.00
MOVL C00112 BC00112 V=166.7 PL=0
REFP 3 C00113 BC00113
CALL JOB:SEARCH-R1
SET P0352 P0006
SFTON P0352
MOVL C00114 BC00114 V=166.7 PL=0
REFP 3 C00115 BC00115
CALL JOB:SEARCH-R1
SET P0352 P0006
SFTON P0352
MOVL C00116 BC00116 V=166.7 PL=0
SFTOF
'------------------------
'W250A P
'------------------------
MOVJ C00117 BC00117 VJ=40.00
MOVL C00118 BC00118 V=166.7 PL=0
REFP 3 C00119 BC00119
CALL JOB:SEARCH-R1
SET P0353 P0006
SFTON P0353
MOVL C00120 BC00120 V=66.7 PL=0
REFP 3 C00121 BC00121
CALL JOB:SEARCH-R1
SET P0353 P0006
SFTON P0353
MOVL C00122 BC00122 V=66.7 PL=0
SFTOF
'------------------------
'W250A L
'------------------------
MOVJ C00123 BC00123 VJ=40.00
MOVL C00124 BC00124 V=166.7 PL=0
REFP 3 C00125 BC00125
CALL JOB:SEARCH-R1
SET P0354 P0006
SFTON P0354
MOVL C00126 BC00126 V=66.7 PL=0
REFP 3 C00127 BC00127
CALL JOB:SEARCH-R1
SET P0354 P0006
SFTON P0354
MOVL C00128 BC00128 V=166.7 PL=0
SFTOF
'------------------------
'W253A P
'------------------------
MOVJ C00129 BC00129 VJ=40.00
MOVL C00130 BC00130 V=166.7 PL=0
REFP 3 C00131 BC00131
CALL JOB:SEARCH-R1
SET P0355 P0006
SFTON P0355
MOVL C00132 BC00132 V=166.7 PL=0
REFP 3 C00133 BC00133
CALL JOB:SEARCH-R1
SET P0355 P0006
SFTON P0355
MOVL C00134 BC00134 V=166.7 PL=0
SFTOF
'------------------------
'W253A L
'------------------------
MOVJ C00135 BC00135 VJ=40.00
MOVL C00136 BC00136 V=166.7 PL=0
REFP 3 C00137 BC00137
CALL JOB:SEARCH-R1
SET P0356 P0006
SFTON P0356
MOVL C00138 BC00138 V=166.7 PL=0
REFP 3 C00139 BC00139
CALL JOB:SEARCH-R1
SET P0356 P0006
SFTON P0356
MOVL C00140 BC00140 V=166.7 PL=0
SFTOF
'------------------------
'W256A P
'------------------------
MOVJ C00141 BC00141 VJ=40.00
MOVL C00142 BC00142 V=166.7 PL=0
REFP 3 C00143 BC00143
CALL JOB:SEARCH-R1
SET P0357 P0006
SFTON P0357
MOVL C00144 BC00144 V=166.7 PL=0
REFP 3 C00145 BC00145
CALL JOB:SEARCH-R1
SET P0357 P0006
SFTON P0357
MOVL C00146 BC00146 V=166.7 PL=0
SFTOF
'------------------------
'W256A L
'------------------------
MOVJ C00147 BC00147 VJ=40.00
MOVL C00148 BC00148 V=166.7 PL=0
REFP 3 C00149 BC00149
CALL JOB:SEARCH-R1
SET P0358 P0006
SFTON P0358
MOVL C00150 BC00150 V=166.7 PL=0
REFP 3 C00151 BC00151
CALL JOB:SEARCH-R1
SET P0358 P0006
SFTON P0358
MOVL C00152 BC00152 V=166.7 PL=0
SFTOF
'------------------------
'W252A P
'------------------------
MOVL C00153 BC00153 V=666.7
MOVL C00154 BC00154 V=166.7 PL=0
REFP 3 C00155 BC00155
CALL JOB:SEARCH-R1
SET P0359 P0006
SFTON P0359
MOVL C00156 BC00156 V=166.7 PL=0
REFP 3 C00157 BC00157
CALL JOB:SEARCH-R1
SET P0359 P0006
SFTON P0359
MOVL C00158 BC00158 V=166.7 PL=0
SFTOF
'------------------------
'W252A L
'------------------------
MOVL C00159 BC00159 V=500.0
MOVL C00160 BC00160 V=166.7 PL=0
REFP 3 C00161 BC00161
CALL JOB:SEARCH-R1
SET P0360 P0006
SFTON P0360
MOVL C00162 BC00162 V=166.7 PL=0
REFP 3 C00163 BC00163
CALL JOB:SEARCH-R1
SET P0360 P0006
SFTON P0360
MOVL C00164 BC00164 V=166.7 PL=0
SFTOF
'------------------------
'W255A
'------------------------
MOVL C00165 BC00165 V=500.0
MOVL C00166 BC00166 V=166.7 PL=0
REFP 3 C00167 BC00167
CALL JOB:SEARCH-R1
SET P0361 P0006
SFTON P0361
MOVL C00168 BC00168 V=166.7 PL=0
REFP 3 C00169 BC00169
CALL JOB:SEARCH-R1
SET P0361 P0006
SFTON P0361
MOVL C00170 BC00170 V=166.7 PL=0
SFTOF
MOVL C00171 BC00171 V=500.0
MOVL C00172 BC00172 V=166.7 PL=0
REFP 3 C00173 BC00173
CALL JOB:SEARCH-R1
SET P0362 P0006
SFTON P0362
MOVL C00174 BC00174 V=166.7 PL=0
REFP 3 C00175 BC00175
CALL JOB:SEARCH-R1
SET P0362 P0006
SFTON P0362
MOVL C00176 BC00176 V=166.7 PL=0
SFTOF
MOVL C00177 BC00177 V=666.7
MOVL C00178 BC00178 V=666.7
MOVL C00179 BC00179 V=666.7
MOVJ C00180 BC00180 VJ=40.00
MOVJ C00181 BC00181 VJ=40.00
COMM MOVJ C00182 BC00182 VJ=40.00
COMM MOVJ C00183 BC00183 VJ=40.00
COMM MOVJ C00184 BC00184 VJ=40.00
COMM MOVJ C00185 BC00185 VJ=40.00
COMM MOVJ C00186 BC00186 VJ=30.00
COMM '------------------------
COMM 'W61.3
COMM '------------------------
COMM MOVL C00187 BC00187 V=500.0
COMM MOVL C00188 BC00188 V=166.7 PL=0
COMM REFP 3 C00189 BC00189
COMM CALL JOB:SEARCH-R1
COMM SET P0400 P0006
COMM SFTON P0400
COMM MOVL C00190 BC00190 V=166.7 PL=0
COMM REFP 3 C00191 BC00191
COMM CALL JOB:SEARCH-R1
COMM SET P0400 P0006
COMM SFTON P0400
COMM MOVL C00192 BC00192 V=166.7 PL=0
COMM SFTOF
COMM 'BELKA PRZEJAZD
COMM MOVL C00193 BC00193 V=333.3
COMM '------------------------
COMM 'W61.5
COMM '------------------------
COMM MOVL C00194 BC00194 V=166.7 PL=0
COMM REFP 3 C00195 BC00195
COMM CALL JOB:SEARCH-R1
COMM SET P0401 P0006
COMM SFTON P0401
COMM MOVL C00196 BC00196 V=166.7 PL=0
COMM REFP 3 C00197 BC00197
COMM CALL JOB:SEARCH-R1
COMM SET P0401 P0006
COMM SFTON P0401
COMM MOVL C00198 BC00198 V=166.7 PL=0
COMM SFTOF
COMM '------------------------
COMM 'W61.7
COMM '------------------------
COMM MOVL C00199 BC00199 V=500.0
COMM MOVL C00200 BC00200 V=166.7 PL=0
COMM REFP 3 C00201 BC00201
COMM CALL JOB:SEARCH-R1
COMM SET P0402 P0006
COMM SFTON P0402
COMM MOVL C00202 BC00202 V=166.7 PL=0
COMM REFP 3 C00203 BC00203
COMM CALL JOB:SEARCH-R1
COMM SET P0402 P0006
COMM SFTON P0402
COMM MOVL C00204 BC00204 V=166.7 PL=0
COMM SFTOF
COMM MOVL C00205 BC00205 V=500.0
COMM '------------------------
COMM 'W61.10
COMM '------------------------
COMM MOVJ C00206 BC00206 VJ=30.00
COMM MOVJ C00207 BC00207 VJ=50.00
COMM MOVJ C00208 BC00208 VJ=50.00
COMM MOVL C00209 BC00209 V=500.0
COMM MOVL C00210 BC00210 V=166.7 PL=0
COMM REFP 3 C00211 BC00211
COMM CALL JOB:SEARCH-R1
COMM SET P0403 P0006
COMM SFTON P0403
COMM MOVL C00212 BC00212 V=166.7 PL=0
COMM REFP 3 C00213 BC00213
COMM CALL JOB:SEARCH-R1
COMM SET P0403 P0006
COMM SFTON P0403
COMM MOVL C00214 BC00214 V=166.7 PL=0
COMM SFTOF
COMM MOVL C00215 BC00215 V=333.3
COMM '------------------------
COMM 'W61.12
COMM '------------------------
COMM MOVL C00216 BC00216 V=666.7
COMM MOVL C00217 BC00217 V=166.7 PL=0
COMM REFP 3 C00218 BC00218
COMM CALL JOB:SEARCH-R1
COMM SET P0404 P0006
COMM SFTON P0404
COMM MOVL C00219 BC00219 V=166.7 PL=0
COMM REFP 3 C00220 BC00220
COMM CALL JOB:SEARCH-R1
COMM SET P0404 P0006
COMM SFTON P0404
COMM MOVL C00221 BC00221 V=166.7 PL=0
COMM SFTOF
COMM '------------------------
COMM 'W61.15
COMM '------------------------
COMM MOVL C00222 BC00222 V=666.7
COMM MOVL C00223 BC00223 V=166.7 PL=0
COMM REFP 3 C00224 BC00224
COMM CALL JOB:SEARCH-R1
COMM SET P0405 P0006
COMM SFTON P0405
COMM MOVL C00225 BC00225 V=166.7 PL=0
COMM REFP 3 C00226 BC00226
COMM CALL JOB:SEARCH-R1
COMM SET P0405 P0006
COMM SFTON P0405
COMM MOVL C00227 BC00227 V=166.7 PL=0
COMM SFTOF
COMM MOVL C00228 BC00228 V=666.7
COMM MOVJ C00229 BC00229 VJ=50.00
COMM MOVJ C00230 BC00230 VJ=50.00
COMM MOVJ C00231 BC00231 VJ=50.00
COMM '------------------------
COMM 'W61.17
COMM '------------------------
COMM MOVL C00232 BC00232 V=416.7
COMM MOVL C00233 BC00233 V=166.7 PL=0
COMM REFP 3 C00234 BC00234
COMM CALL JOB:SEARCH-R1
COMM SET P0406 P0006
COMM SFTON P0406
COMM MOVL C00235 BC00235 V=166.7 PL=0
COMM REFP 3 C00236 BC00236
COMM CALL JOB:SEARCH-R1
COMM SET P0406 P0006
COMM SFTON P0406
COMM MOVL C00237 BC00237 V=166.7 PL=0
COMM SFTOF
COMM MOVL C00238 BC00238 V=333.3
COMM '------------------------
COMM 'W61.20
COMM '------------------------
COMM MOVL C00239 BC00239 V=666.7
COMM MOVL C00240 BC00240 V=166.7 PL=0
COMM REFP 3 C00241 BC00241
COMM CALL JOB:SEARCH-R1
COMM SET P0407 P0006
COMM SFTON P0407
COMM MOVL C00242 BC00242 V=166.7 PL=0
COMM REFP 3 C00243 BC00243
COMM CALL JOB:SEARCH-R1
COMM SET P0407 P0006
COMM SFTON P0407
COMM MOVL C00244 BC00244 V=166.7 PL=0
COMM SFTOF
COMM '------------------------
COMM 'W61.23
COMM '------------------------
COMM MOVL C00245 BC00245 V=500.0
COMM MOVL C00246 BC00246 V=166.7 PL=0
COMM REFP 3 C00247 BC00247
COMM CALL JOB:SEARCH-R1
COMM SET P0408 P0006
COMM SFTON P0408
COMM MOVL C00248 BC00248 V=166.7 PL=0
COMM REFP 3 C00249 BC00249
COMM CALL JOB:SEARCH-R1
COMM SET P0408 P0006
COMM SFTON P0408
COMM MOVL C00250 BC00250 V=166.7 PL=0
COMM SFTOF
COMM MOVL C00251 BC00251 V=333.3
COMM MOVL C00252 BC00252 V=666.7
COMM MOVL C00253 BC00253 V=666.7
COMM '------------------------
COMM 'W61.25
COMM '------------------------
COMM MOVL C00254 BC00254 V=500.0
COMM MOVL C00255 BC00255 V=166.7 PL=0
COMM REFP 3 C00256 BC00256
COMM CALL JOB:SEARCH-R1
COMM SET P0409 P0006
COMM SFTON P0409
COMM MOVL C00257 BC00257 V=166.7 PL=0
COMM REFP 3 C00258 BC00258
COMM CALL JOB:SEARCH-R1
COMM SET P0409 P0006
COMM SFTON P0409
COMM MOVL C00259 BC00259 V=166.7 PL=0
COMM SFTOF
COMM MOVL C00260 BC00260 V=666.7
COMM MOVJ C00261 BC00261 VJ=50.00
COMM MOVJ C00262 BC00262 VJ=50.00
COMM GETE D040 P0409 (1)
COMM GETE D041 P0409 (2)
COMM GETE D042 P0409 (3)
COMM SETE P0410 (1) D040
COMM SETE P0410 (2) D041
COMM SETE P0410 (3) D042
COMM '------------------------
COMM 'W61.30
COMM '------------------------
COMM MOVL C00263 BC00263 V=500.0
COMM MOVL C00264 BC00264 V=166.7 PL=0
COMM REFP 3 C00265 BC00265
COMM CALL JOB:SEARCH-R1
COMM SET P0411 P0006
COMM SFTON P0411
COMM MOVL C00266 BC00266 V=166.7 PL=0
COMM REFP 3 C00267 BC00267
COMM CALL JOB:SEARCH-R1
COMM SET P0411 P0006
COMM SFTON P0411
COMM MOVL C00268 BC00268 V=166.7 PL=0
COMM SFTOF
COMM MOVL C00269 BC00269 V=666.7
COMM MOVJ C00270 BC00270 VJ=50.00
MOVJ C00271 BC00271 VJ=70.00
CALL JOB:FRONT_SEARCH_-90ST-2_5540
MOVJ C00272 BC00272 VJ=60.00
MOVJ C00273 BC00273 VJ=50.00
MOVJ C00274 BC00274 VJ=50.00
MOVL C00275 BC00275 V=666.7
MOVJ C00276 BC00276 VJ=30.00
'------------------------
'W65.3
'------------------------
SFTON P0300
MOVL C00277 BC00277 V=333.3
MOVL C00278 BC00278 V=166.7 PL=0
MACRO1 MJ#(0) ARGF10
ARCON
MOVL C00279 BC00279 V=10.8
ARCOF
MOVL C00280 BC00280 V=166.7
SFTOF
'------------------------
'W65.5
'------------------------
SFTON P0301
MOVL C00281 BC00281 V=666.7
MOVL C00282 BC00282 V=166.7 PL=0
MACRO1 MJ#(0) ARGF9
ARCON
MOVL C00283 BC00283 V=8.3
ARCOF
MOVL C00284 BC00284 V=166.7
SFTOF
MOVL C00285 BC00285 V=500.0
MOVL C00286 BC00286 V=666.7
MOVJ C00287 BC00287 VJ=40.00
COMM MOVJ C00288 BC00288 VJ=60.00
COMM '::::::::::::::::::::::::::::::::
COMM '::::::::::::::::::::::::::::::::
COMM '::::::::::::::::::::::::::::::::
COMM '::::::::::::::::::::::::::::::::
COMM '::::::::::::::::::::::::::::::::
COMM MOVJ C00289 BC00289 VJ=50.00
COMM MOVJ C00290 BC00290 VJ=50.00
COMM MOVJ C00291 BC00291 VJ=40.00
COMM MOVJ C00292 BC00292 VJ=40.00
COMM MOVJ C00293 BC00293 VJ=40.00
COMM MOVJ C00294 BC00294 VJ=40.00
COMM MOVL C00295 BC00295 V=666.7
COMM '------------------------
COMM 'W61.3
COMM '------------------------
COMM SFTON P0400
COMM ARCOF
COMM MOVL C00296 BC00296 V=500.0
COMM SFTOF
COMM 'BELKA PRZEJAZD
COMM '------------------------
COMM 'W61.5
COMM '------------------------
COMM SFTON P0401
COMM MOVL C00297 BC00297 V=666.7
COMM MOVL C00298 BC00298 V=166.7 PL=0
COMM MACRO1 MJ#(0) ARGF24
COMM ARCON
COMM MOVL C00299 BC00299 V=7.5
COMM ARCOF
COMM MOVL C00300 BC00300 V=250.0
COMM SFTOF
COMM MOVL C00301 BC00301 V=500.0
COMM MOVJ C00302 BC00302 VJ=40.00
COMM MOVJ C00303 BC00303 VJ=40.00
COMM MOVJ C00304 BC00304 VJ=50.00
COMM MOVJ C00305 BC00305 VJ=50.00
MOVJ C00306 BC00306 VJ=50.00
MOVJ C00307 BC00307 VJ=50.00
MOVL C00308 BC00308 V=666.7
'------------------------
'W250A
'------------------------
SFTON P0354
MOVL C00309 BC00309 V=666.7
MOVL C00310 BC00310 V=166.7 PL=0
MACRO1 MJ#(0) ARGF9
ARCON
SFTOF
SFTON P0353
MOVL C00311 BC00311 V=11.7
ARCOF
MOVL C00312 BC00312 V=333.3
SFTOF
MOVJ C00313 BC00313 VJ=50.00
MOVJ C00314 BC00314 VJ=60.00
MOVJ C00315 BC00315 VJ=40.00
MOVJ C00316 BC00316 VJ=50.00
MOVJ C00317 BC00317 VJ=40.00
MOVJ C00318 BC00318 VJ=30.00
MOVJ C00319 BC00319 VJ=15.00
'------------------------
'W65.7
'------------------------
SFTON P0302
MOVL C00320 BC00320 V=833.3
MOVL C00321 BC00321 V=166.7 PL=0
MACRO1 MJ#(0) ARGF10
ARCON
MOVL C00322 BC00322 V=10.8
ARCOF
MOVL C00323 BC00323 V=166.7
SFTOF
'------------------------
'W65.10
'------------------------
SFTON P0303
MOVL C00324 BC00324 V=666.7
MOVL C00325 BC00325 V=166.7 PL=0
ARCON
MOVL C00326 BC00326 V=10.8
ARCOF
MOVL C00327 BC00327 V=166.7
SFTOF
MOVL C00328 BC00328 V=333.3
MOVL C00329 BC00329 V=666.7
MOVJ C00330 BC00330 VJ=30.00
MOVJ C00331 BC00331 VJ=30.00
MOVJ C00332 BC00332 VJ=30.00
MOVJ C00333 BC00333 VJ=50.00
COMM '::::::::::::::::::::::::::::::::
COMM '::::::::::::::::::::::::::::::::
COMM '------------------------
COMM 'W61.7
COMM '------------------------
COMM '::::::::::::::::::::::::::::::::
COMM '::::::::::::::::::::::::::::::::
COMM MOVJ C00334 BC00334 VJ=30.00
COMM MOVJ C00335 BC00335 VJ=30.00
COMM MOVJ C00336 BC00336 VJ=40.00
COMM SFTON P0402
COMM MOVL C00337 BC00337 V=500.0
COMM MOVL C00338 BC00338 V=166.7 PL=0
COMM MACRO1 MJ#(0) ARGF24
COMM ARCON
COMM MOVL C00339 BC00339 V=7.5
COMM ARCOF
COMM MOVL C00340 BC00340 V=250.0
COMM SFTOF
COMM MOVJ C00341 BC00341 VJ=30.00
COMM MOVJ C00342 BC00342 VJ=40.00
COMM MOVJ C00343 BC00343 VJ=50.00
COMM '------------------------
COMM 'W61.10
COMM '------------------------
COMM SFTON P0403
COMM MOVL C00344 BC00344 V=500.0
COMM MOVL C00345 BC00345 V=166.7 PL=0
COMM MACRO1 MJ#(0) ARGF24
COMM ARCON
COMM MOVL C00346 BC00346 V=7.5
COMM ARCOF
COMM MOVL C00347 BC00347 V=250.0
COMM SFTOF
COMM MOVL C00348 BC00348 V=500.0
COMM MOVL C00349 BC00349 V=666.7
COMM MOVL C00350 BC00350 V=666.7
COMM MOVJ C00351 BC00351 VJ=50.00
COMM MOVJ C00352 BC00352 VJ=50.00
COMM MOVJ C00353 BC00353 VJ=50.00
COMM '::::::::::::::::::::::::
COMM '::::::::::::::::::::::::
COMM '::::::::::::::::::::::::
COMM '::::::::::::::::::::::::
COMM '::::::::::::::::::::::::
COMM '::::::::::::::::::::::::
COMM '::::::::::::::::::::::::
MOVJ C00354 BC00354 VJ=50.00
MOVJ C00355 BC00355 VJ=50.00
MOVJ C00356 BC00356 VJ=50.00
'------------------------
'W251B
'------------------------
MOVL C00357 BC00357 V=500.0
MOVL C00358 BC00358 V=500.0
SFTON P0350
MOVL C00359 BC00359 V=166.7 PL=0
MACRO1 MJ#(0) ARGF9
ARCON
SFTOF
SFTON P0349
MOVL C00360 BC00360 V=11.3
MOVL C00361 BC00361 V=11.3
ARCOF
MOVL C00362 BC00362 V=333.3
SFTOF
MOVJ C00363 BC00363 VJ=50.00
MOVJ C00364 BC00364 VJ=50.00
MOVJ C00365 BC00365 VJ=10.00
MOVJ C00366 BC00366 VJ=50.00
MOVJ C00367 BC00367 VJ=50.00
MOVJ C00368 BC00368 VJ=25.00
MOVJ C00369 BC00369 VJ=20.00
MOVJ C00370 BC00370 VJ=20.00
'------------------------
'W65.12
'------------------------
SFTON P0304
MOVL C00371 BC00371 V=333.3
MOVL C00372 BC00372 V=166.7 PL=0
MACRO1 MJ#(0) ARGF10
ARCON
MOVL C00373 BC00373 V=10.8
ARCOF
MOVL C00374 BC00374 V=166.7
SFTOF
'------------------------
'W65.15
'------------------------
SFTON P0305
MOVL C00375 BC00375 V=666.7
MOVL C00376 BC00376 V=166.7 PL=0
MACRO1 MJ#(0) ARGF9
ARCON
MOVL C00377 BC00377 V=10.8
ARCOF
MOVL C00378 BC00378 V=200.0
SFTOF
MOVL C00379 BC00379 V=250.0
MOVL C00380 BC00380 V=416.7
MOVL C00381 BC00381 V=666.7
COMM MOVJ C00382 BC00382 VJ=50.00
COMM MOVJ C00383 BC00383 VJ=50.00
COMM '::::::::::::::::::::::::
COMM '::::::::::::::::::::::::
COMM '::::::::::::::::::::::::
COMM '::::::::::::::::::::::::
COMM '::::::::::::::::::::::::
COMM '::::::::::::::::::::::::
COMM '::::::::::::::::::::::::
COMM MOVJ C00384 BC00384 VJ=50.00
COMM MOVJ C00385 BC00385 VJ=50.00
COMM MOVJ C00386 BC00386 VJ=50.00
COMM '::::::::::::::::::::::::::::::::
COMM '::::::::::::::::::::::::::::::::
COMM '------------------------
COMM 'W61.12
COMM '------------------------
COMM '::::::::::::::::::::::::::::::::
COMM '::::::::::::::::::::::::::::::::
COMM MOVL C00387 BC00387 V=833.3
COMM MOVL C00388 BC00388 V=666.7
COMM MOVL C00389 BC00389 V=500.0
COMM SFTON P0404
COMM MOVL C00390 BC00390 V=166.7 PL=0
COMM MACRO1 MJ#(0) ARGF24
COMM ARCON
COMM MOVL C00391 BC00391 V=6.7
COMM ARCOF
COMM MOVL C00392 BC00392 V=333.3
COMM SFTOF
COMM MOVL C00393 BC00393 V=500.0
COMM MOVL C00394 BC00394 V=666.7
COMM '------------------------
COMM 'W61.15
COMM '------------------------
COMM SFTON P0405
COMM MOVL C00395 BC00395 V=666.7
COMM MOVL C00396 BC00396 V=166.7 PL=0
COMM MACRO1 MJ#(0) ARGF24
COMM ARCON
COMM MOVL C00397 BC00397 V=6.7
COMM ARCOF
COMM MOVL C00398 BC00398 V=250.0
COMM SFTOF
COMM MOVJ C00399 BC00399 VJ=40.00
COMM MOVJ C00400 BC00400 VJ=40.00
COMM MOVJ C00401 BC00401 VJ=40.00
COMM MOVJ C00402 BC00402 VJ=40.00
COMM '::::::::::::::::::::::::
COMM '::::::::::::::::::::::::
COMM '::::::::::::::::::::::::
COMM '::::::::::::::::::::::::
COMM '::::::::::::::::::::::::
COMM '::::::::::::::::::::::::
COMM '::::::::::::::::::::::::
COMM MOVJ C00403 BC00403 VJ=40.00
COMM MOVJ C00404 BC00404 VJ=40.00
COMM '------------------------
COMM 'W252B
COMM '------------------------
SFTON P0359
MOVL C00405 BC00405 V=666.7
MOVL C00406 BC00406 V=166.7 PL=0
MACRO1 MJ#(0) ARGF9
ARCON
SFTOF
SFTON P0358
MOVL C00407 BC00407 V=10.8
ARCOF
MOVL C00408 BC00408 V=250.0
SFTOF
MOVJ C00409 BC00409 VJ=50.00
MOVJ C00410 BC00410 VJ=50.00
MOVJ C00411 BC00411 VJ=60.00
MOVJ C00412 BC00412 VJ=40.00
MOVJ C00413 BC00413 VJ=30.00
MOVL C00414 BC00414 V=500.0
MOVL C00415 BC00415 V=333.3
'------------------------
'W65.17
'------------------------
SFTON P0306
MOVL C00416 BC00416 V=333.3
MOVL C00417 BC00417 V=166.7 PL=0
MACRO1 MJ#(0) ARGF10
ARCON
MOVL C00418 BC00418 V=10.8
ARCOF
MOVL C00419 BC00419 V=166.7
SFTOF
MOVL C00420 BC00420 V=333.3
MOVL C00421 BC00421 V=500.0
MOVL C00422 BC00422 V=500.0
MOVJ C00423 BC00423 VJ=40.00
COMM MOVJ C00424 BC00424 VJ=60.00
COMM MOVJ C00425 BC00425 VJ=60.00
COMM '::::::::::::::::::::::::
COMM '::::::::::::::::::::::::
COMM '::::::::::::::::::::::::
COMM '::::::::::::::::::::::::
COMM '::::::::::::::::::::::::
COMM '::::::::::::::::::::::::
COMM '::::::::::::::::::::::::
COMM MOVJ C00426 BC00426 VJ=60.00
COMM '::::::::::::::::::::::::::::::::
COMM '::::::::::::::::::::::::::::::::
COMM '------------------------
COMM 'W61.17
COMM '------------------------
COMM '::::::::::::::::::::::::::::::::
COMM '::::::::::::::::::::::::::::::::
COMM SFTON P0406
COMM MOVJ C00427 BC00427 VJ=40.00
COMM MOVL C00428 BC00428 V=500.0
COMM MOVL C00429 BC00429 V=166.7 PL=0
COMM MACRO1 MJ#(0) ARGF24
COMM ARCON
COMM MOVL C00430 BC00430 V=6.7
COMM ARCOF
COMM MOVL C00431 BC00431 V=333.3
COMM SFTOF
COMM MOVJ C00432 BC00432 VJ=30.00
COMM MOVJ C00433 BC00433 VJ=40.00
COMM MOVJ C00434 BC00434 VJ=50.00
COMM '------------------------
COMM 'W253A
'------------------------
COMM MOVJ C00435 BC00435 VJ=50.00
MOVJ C00436 BC00436 VJ=50.00
SFTON P0356
MOVL C00437 BC00437 V=500.0
MOVL C00438 BC00438 V=500.0
MOVL C00439 BC00439 V=166.7 PL=0
MACRO1 MJ#(0) ARGF9
ARCON
SFTOF
SFTON P0355
MOVL C00440 BC00440 V=11.3
ARCOF
MOVL C00441 BC00441 V=333.3
SFTOF
MOVJ C00442 BC00442 VJ=50.00
'------------------------
'W65.20
'------------------------
COMM MOVJ C00443 BC00443 VJ=50.00
COMM MOVJ C00444 BC00444 VJ=50.00
COMM MOVJ C00445 BC00445 VJ=50.00
COMM '::::::::::::::::::::::::
COMM '::::::::::::::::::::::::
COMM '::::::::::::::::::::::::
COMM '::::::::::::::::::::::::
COMM '::::::::::::::::::::::::
COMM '::::::::::::::::::::::::
COMM '::::::::::::::::::::::::
COMM MOVJ C00446 BC00446 VJ=40.00
COMM MOVJ C00447 BC00447 VJ=40.00
COMM '::::::::::::::::::::::::::::::::
COMM '::::::::::::::::::::::::::::::::
COMM '------------------------
COMM 'W61.20
COMM '------------------------
COMM '::::::::::::::::::::::::::::::::
COMM '::::::::::::::::::::::::::::::::
COMM SFTON P0407
COMM MOVL C00448 BC00448 V=666.7
COMM MOVL C00449 BC00449 V=333.3
COMM MOVL C00450 BC00450 V=166.7 PL=0
COMM MACRO1 MJ#(0) ARGF24
COMM ARCON
COMM MOVL C00451 BC00451 V=6.7
COMM ARCOF
COMM MOVL C00452 BC00452 V=250.0
COMM SFTOF
COMM '::::::::::::::::::::::::
COMM '::::::::::::::::::::::::
COMM '::::::::::::::::::::::::
COMM '::::::::::::::::::::::::
COMM '::::::::::::::::::::::::
COMM MOVL C00453 BC00453 V=500.0
COMM MOVJ C00454 BC00454 VJ=50.00
COMM MOVJ C00455 BC00455 VJ=50.00
COMM MOVJ C00456 BC00456 VJ=50.00
COMM '------------------------
COMM 'W254A
COMM '------------------------
COMM MOVJ C00457 BC00457 VJ=50.00
MOVJ C00458 BC00458 VJ=50.00
SFTON P0352
MOVL C00459 BC00459 V=666.7
MOVL C00460 BC00460 V=500.0
MOVL C00461 BC00461 V=250.0 PL=0
MACRO1 MJ#(0) ARGF9
ARCON
SFTOF
SFTON P0351
MOVL C00462 BC00462 V=11.2
ARCOF
MOVL C00463 BC00463 V=333.3
MOVL C00464 BC00464 V=666.7
SFTOF
COMM MOVJ C00465 BC00465 VJ=50.00
COMM MOVJ C00466 BC00466 VJ=80.00
COMM MOVJ C00467 BC00467 VJ=50.00
MOVJ C00468 BC00468 VJ=50.00
MOVJ C00469 BC00469 VJ=30.00
MOVL C00470 BC00470 V=666.7
'------------------------
'W65.23
'------------------------
SFTON P0308
MOVL C00471 BC00471 V=333.3
MOVL C00472 BC00472 V=166.7
MOVL C00473 BC00473 V=166.7 PL=0
MACRO1 MJ#(0) ARGF10
ARCON
MOVL C00474 BC00474 V=10.8
ARCOF
MOVL C00475 BC00475 V=250.0
SFTOF
'------------------------
'W65.25
'------------------------
SFTON P0309
MOVL C00476 BC00476 V=666.7
MOVL C00477 BC00477 V=166.7
MOVL C00478 BC00478 V=166.7 PL=0
ARCON
MOVL C00479 BC00479 V=10.8
ARCOF
MOVL C00480 BC00480 V=250.0
SFTOF
MOVL C00481 BC00481 V=250.0
MOVL C00482 BC00482 V=500.0
MOVL C00483 BC00483 V=666.7
MOVL C00484 BC00484 V=666.7
MOVJ C00485 BC00485 VJ=40.00
MOVJ C00486 BC00486 VJ=40.00
MOVJ C00487 BC00487 VJ=50.00
COMM '::::::::::::::::::::::::
COMM '::::::::::::::::::::::::
COMM '::::::::::::::::::::::::
COMM '::::::::::::::::::::::::
COMM '::::::::::::::::::::::::
COMM '::::::::::::::::::::::::
COMM '::::::::::::::::::::::::
COMM MOVJ C00488 BC00488 VJ=50.00
COMM MOVJ C00489 BC00489 VJ=50.00
COMM MOVJ C00490 BC00490 VJ=50.00
COMM '::::::::::::::::::::::::::::::::
COMM '::::::::::::::::::::::::::::::::
COMM '------------------------
COMM 'W61.23
COMM '------------------------
COMM '::::::::::::::::::::::::::::::::
COMM '::::::::::::::::::::::::::::::::
COMM SFTON P0408
COMM MOVL C00491 BC00491 V=500.0
COMM MOVL C00492 BC00492 V=666.7
COMM MOVL C00493 BC00493 V=166.7 PL=0
COMM MACRO1 MJ#(0) ARGF24
COMM ARCON
COMM MOVL C00494 BC00494 V=8.3
COMM ARCOF
COMM MOVL C00495 BC00495 V=250.0
COMM SFTOF
COMM MOVL C00496 BC00496 V=666.7
COMM '------------------------
COMM 'W61.25
COMM '------------------------
COMM SFTON P0409
COMM MOVL C00497 BC00497 V=500.0
COMM MOVL C00498 BC00498 V=166.7 PL=0
COMM MACRO1 MJ#(0) ARGF24
COMM ARCON
COMM MOVL C00499 BC00499 V=8.3
COMM ARCOF
COMM MOVL C00500 BC00500 V=166.7
COMM SFTOF
COMM MOVL C00501 BC00501 V=500.0
COMM MOVJ C00502 BC00502 VJ=20.00
COMM '::::::::::::::::::::::::
COMM '::::::::::::::::::::::::
COMM '::::::::::::::::::::::::
COMM '::::::::::::::::::::::::
COMM '::::::::::::::::::::::::
COMM MOVJ C00503 BC00503 VJ=50.00
COMM MOVJ C00504 BC00504 VJ=50.00
MOVJ C00505 BC00505 VJ=40.00
'------------------------
'W255A
MOVL C00506 BC00506 V=500.0
MOVL C00507 BC00507 V=666.7
SFTON P0361
MOVL C00508 BC00508 V=166.7 PL=0
MACRO1 MJ#(0) ARGF9
ARCON
SFTON P0362
MOVL C00509 BC00509 V=11.2
MOVL C00510 BC00510 V=10.8
ARCOF
MOVL C00511 BC00511 V=333.3
SFTOF
MOVL C00512 BC00512 V=666.7
MOVL C00513 BC00513 V=666.7
MOVL C00514 BC00514 V=666.7
MOVJ C00515 BC00515 VJ=50.00
MOVJ C00516 BC00516 VJ=70.00
MOVJ C00517 BC00517 VJ=70.00
MOVJ C00518 BC00518 VJ=50.00
MOVJ C00519 BC00519 VJ=50.00
MOVJ C00520 BC00520 VJ=50.00
MOVL C00521 BC00521 V=500.0
'------------------------
'W31.28
'------------------------
MOVL C00522 BC00522 V=333.3
MOVL C00523 BC00523 V=333.3
MACRO1 MJ#(0) ARGF10
SFTON P0311
MOVL C00524 BC00524 V=166.7
ARCON
MOVL C00525 BC00525 V=10.8
ARCOF
MOVL C00526 BC00526 V=250.0
MOVL C00527 BC00527 V=250.0
MOVL C00528 BC00528 V=200.0
ARCON
MOVL C00529 BC00529 V=10.8
ARCOF
MOVL C00530 BC00530 V=166.7
MOVL C00531 BC00531 V=333.3
SFTOF
SFTON P0312
MOVL C00532 BC00532 V=166.7
ARCON
MOVL C00533 BC00533 V=10.8
ARCOF
MOVL C00534 BC00534 V=166.7
MOVL C00535 BC00535 V=166.7
MOVL C00536 BC00536 V=166.7
ARCON
MOVL C00537 BC00537 V=10.8
ARCOF
'------------------------
SFTOF
MOVL C00538 BC00538 V=250.0
MOVL C00539 BC00539 V=416.7
MOVL C00540 BC00540 V=500.0
MOVL C00541 BC00541 V=500.0
MOVL C00542 BC00542 V=666.7
MOVJ C00543 BC00543 VJ=25.00
COMM '::::::::::::::::::::::::
COMM '::::::::::::::::::::::::
COMM '::::::::::::::::::::::::
COMM '::::::::::::::::::::::::
COMM '::::::::::::::::::::::::
COMM '::::::::::::::::::::::::
COMM '::::::::::::::::::::::::
COMM MOVJ C00544 BC00544 VJ=20.00
COMM MOVJ C00545 BC00545 VJ=30.00
COMM '::::::::::::::::::::::::::::::::
COMM '::::::::::::::::::::::::::::::::
COMM '------------------------
COMM 'W61.30
COMM '------------------------
COMM '::::::::::::::::::::::::::::::::
COMM '::::::::::::::::::::::::::::::::
COMM SFTON P0411
COMM MOVL C00546 BC00546 V=500.0
COMM MOVL C00547 BC00547 V=166.7 PL=0
COMM MACRO1 MJ#(0) ARGF24
COMM ARCON
COMM MOVL C00548 BC00548 V=7.5
COMM ARCOF
COMM MOVL C00549 BC00549 V=250.0
COMM MOVL C00550 BC00550 V=500.0
COMM MOVL C00551 BC00551 V=166.7 PL=0
COMM MACRO1 MJ#(0) ARGF24
COMM ARCON
COMM MOVL C00552 BC00552 V=7.5
COMM ARCOF
COMM MOVL C00553 BC00553 V=250.0
COMM SFTOF
COMM MOVL C00554 BC00554 V=500.0
COMM SFTOF
COMM MOVL C00555 BC00555 V=500.0
COMM MOVJ C00556 BC00556 VJ=25.00
MOVJ C00557 BC00557 VJ=50.00
MOVJ C00558 BC00558 VJ=50.00
MOVJ C00559 BC00559 VJ=60.00
'------------------------
'W256A
'------------------------
MOVJ C00560 BC00560 VJ=60.00
MOVJ C00561 BC00561 VJ=60.00
SFTON P0358
MOVL C00562 BC00562 V=666.7
MOVL C00563 BC00563 V=250.0
MOVL C00564 BC00564 V=166.7 PL=0
MACRO1 MJ#(0) ARGF9
ARCON
SFTOF
SFTON P0357
MOVL C00565 BC00565 V=11.2
ARCOF
MOVL C00566 BC00566 V=333.3
SFTOF
MOVJ C00567 BC00567 VJ=50.00
MOVJ C00568 BC00568 VJ=50.00
CALL JOB:FRONT_WELD_-90ST-2_5540
CALL JOB:MOVE_OUT_OF_TUNNEL
END
